(* CoDeSys 2.3.9.62 project: Ascensor_con_memoria_puerta_emergencia.pro *)
(* Libraries: Standard.lib 2.6.14 10:37:46, IecSfc.lib 2.6.14 11:37:46 *)

(* Global variable list: Global_Variables *)
VAR_GLOBAL
   (*Entradas *)

      (* Sensores de posición en plantas *)
      S0_1: BOOL;
      S1_1: BOOL;
      S2_1: BOOL;
      S3_1: BOOL;
      S0_2: BOOL;
      S1_2: BOOL;
      S2_2: BOOL;
      S3_2: BOOL;
      (* Pulsadores de llamadas en planta *)
      P0: BOOL;
      P1: BOOL;
      P2: BOOL;
      P3: BOOL;
    (* Pulsadores en cabina  *)
      C0_1: BOOL;
      C1_1: BOOL;
      C2_1: BOOL;
      C3_1: BOOL;
      C0_2: BOOL;
      C1_2: BOOL;
      C2_2: BOOL;
      C3_2: BOOL;
   (*Salidas *)
      Motor_arriba_1 : BOOL;
      Motor_Abajo_1 : BOOL;
     Motor_arriba_2 : BOOL;
      Motor_Abajo_2 : BOOL;
   (* luces asociadas a los pulsadores. Se usarán
        si se quiere implementar memoria de llamada *)
     LuzP0:BOOL;
     LuzP1:BOOL;
     LuzP2:BOOL;
     LuzP3:BOOL;
     LuzC0_1:BOOL;
     LuzC1_1:BOOL;
     LuzC2_1:BOOL;
     LuzC3_1:BOOL;
     LuzC0_2:BOOL;
     LuzC1_2:BOOL;
     LuzC2_2:BOOL;
     LuzC3_2:BOOL;
(* otras variables*)
	Emergencia: BOOL;
	EmerBTN:BOOL;
	LuzEmer:BOOL;
	Rearme:BOOL;
	puerta:BOOL;
END_VAR

(* POU PLC_PRG, ST *)
PROGRAM PLC_PRG
VAR
END_VAR
Movimiento1;
Ascensor;
END_PROGRAM

(* POU Movimiento1, ST *)
PROGRAM Movimiento1
VAR
    pos1:INT:=0;
END_VAR
IF (Motor_arriba_1 AND pos1>=-240) THEN
   pos1:=pos1-2;
END_IF


IF (Motor_abajo_1 AND pos1<=-2) THEN
   pos1:=pos1+2;
END_IF

IF (pos1>=0 AND pos1<=2) THEN
  S0_1:=TRUE;
ELSE
  S0_1:=FALSE;
END_IF

IF (pos1>=-78 AND pos1<=-74) THEN
  S1_1:=TRUE;
ELSE
  S1_1:=FALSE;
END_IF

IF (pos1>=-156 AND pos1<=-152) THEN
  S2_1:=TRUE;
ELSE
  S2_1:=FALSE;
END_IF

IF (pos1>=-242 AND pos1<=-240) THEN
  S3_1:=TRUE;
ELSE
  S3_1:=FALSE;
END_IF
END_PROGRAM

(* POU Ascensor, SFC *)
PROGRAM Ascensor
VAR
	CicloInicial: BOOL := TRUE;
	luzInt: ARRAY [0..3]  OF BOOL;
	luzext: ARRAY [0..3]  OF BOOL;
	cola: ARRAY [0..4]  OF  BOOL; (* Si la posicion i está a true hay que ir a esa planta *)
	Sentido: BOOL:=TRUE;
	PlantaActual:INT:=0;
	encontrado:BOOL; (* Intero a bool*)
	PD:PlantaDec;
	i: INT; (*interno a seleccion*)
	FRear: F_TRIG;
	REmer: R_TRIG;
	PP: PulsaPlanta;
END_VAR
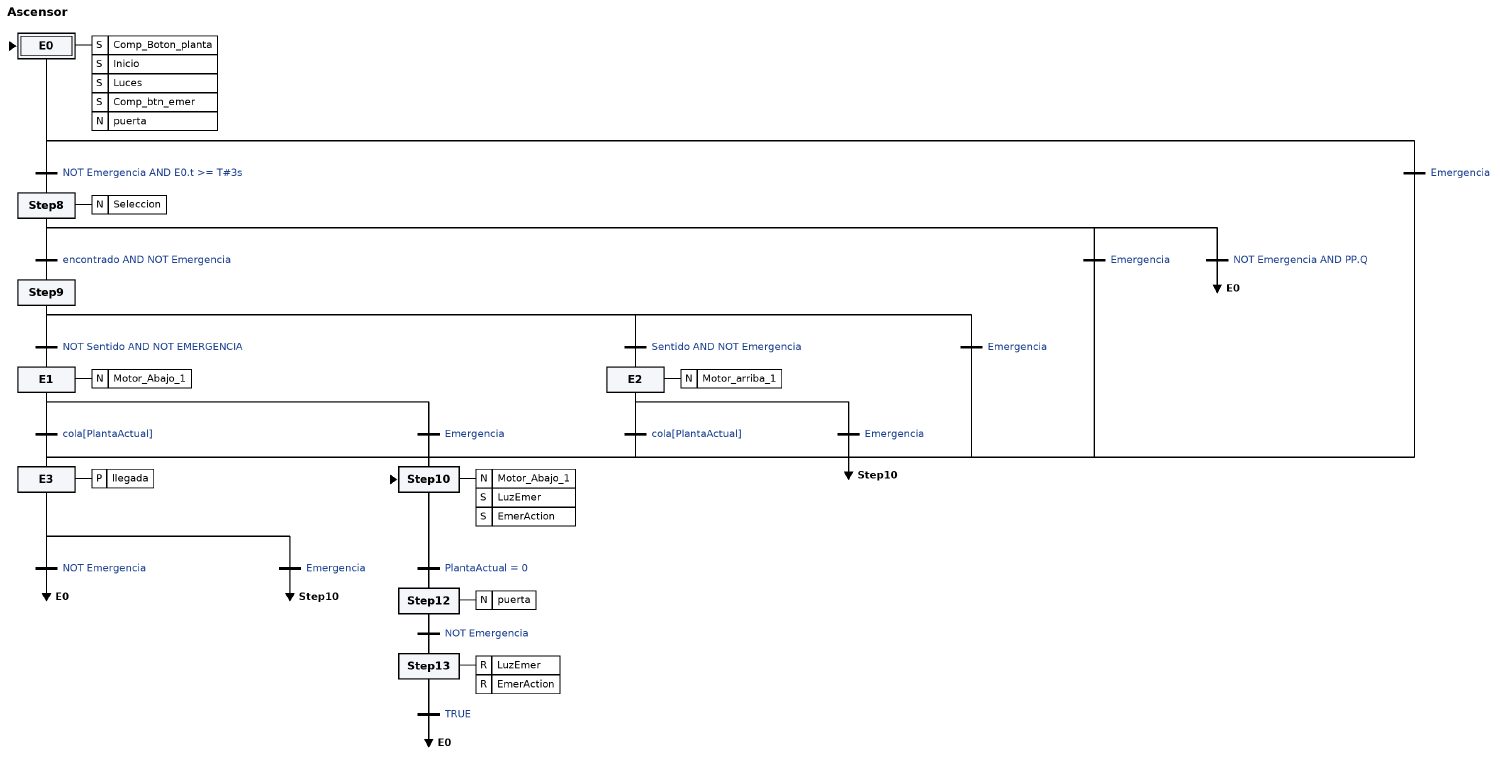
INITIAL_STEP E0:
	Comp_Boton_planta(S);
	Inicio(S);
	Luces(S);
	Comp_btn_emer(S);
	puerta(N);
END_STEP
TRANSITION FROM E0 TO Step8 := NOT Emergencia AND E0.t >= T#3s;
END_TRANSITION
TRANSITION FROM E0 TO Step10 := Emergencia;
END_TRANSITION
STEP Step8:
	Seleccion(N);
END_STEP
TRANSITION FROM Step8 TO Step9 := encontrado AND NOT Emergencia;
END_TRANSITION
TRANSITION FROM Step8 TO Step10 := Emergencia;
END_TRANSITION
TRANSITION FROM Step8 TO E0 := NOT Emergencia AND PP.Q;
END_TRANSITION
STEP Step9:
END_STEP
TRANSITION FROM Step9 TO E1 := NOT Sentido AND NOT EMERGENCIA;
END_TRANSITION
TRANSITION FROM Step9 TO E2 := Sentido AND NOT Emergencia;
END_TRANSITION
TRANSITION FROM Step9 TO Step10 := Emergencia;
END_TRANSITION
STEP E1:
	Motor_Abajo_1(N);
END_STEP
TRANSITION FROM E1 TO E3 := cola[PlantaActual];
END_TRANSITION
TRANSITION FROM E1 TO Step10 := Emergencia;
END_TRANSITION
STEP Step10:
	Motor_Abajo_1(N);
	LuzEmer(S);
	EmerAction(S);
END_STEP
TRANSITION FROM Step10 TO Step12 := PlantaActual = 0;
END_TRANSITION
STEP Step12:
	puerta(N);
END_STEP
TRANSITION FROM Step12 TO Step13 := NOT Emergencia;
END_TRANSITION
STEP Step13:
	LuzEmer(R);
	EmerAction(R);
END_STEP
TRANSITION FROM Step13 TO E0 := TRUE;
END_TRANSITION
STEP E2:
	Motor_arriba_1(N);
END_STEP
TRANSITION FROM E2 TO E3 := cola[PlantaActual];
END_TRANSITION
TRANSITION FROM E2 TO Step10 := Emergencia;
END_TRANSITION
STEP E3:
	llegada(P);
END_STEP
TRANSITION FROM E3 TO E0 := NOT Emergencia;
END_TRANSITION
TRANSITION FROM E3 TO Step10 := Emergencia;
END_TRANSITION
END_PROGRAM
ACTION Comp_Boton_planta:
(* Se encarga de  la  pulsacion de los botones  *)
(* no se puede añadir una planta a la memoria si ya estoy parado  en ella o hay una emergencia *)
IF NOT ( Emergencia OR (S0_1 AND NOT Motor_Abajo_1 AND NOT Motor_arriba_1) )AND (C0_1 OR  P0) THEN
cola[0]:= TRUE;
luzint[0]:= C0_1 OR luzInt[0];
luzext[0]:= P0 OR luzext[0];
ELSIF NOT( Emergencia OR (S1_1 AND NOT Motor_Abajo_1 AND NOT Motor_arriba_1)) AND (C1_1 OR  P1) THEN
cola[1]:= TRUE;
luzint[1]:= C1_1 OR luzInt[1];
luzext[1]:= P1 OR luzext[1];
ELSIF NOT( Emergencia OR (S2_1 AND NOT Motor_Abajo_1 AND NOT Motor_arriba_1) ) AND (C2_1 OR  P2) THEN
cola[2]:= TRUE;
luzint[2]:= C2_1 OR luzInt[2];
luzext[2]:= P2 OR luzext[2];
ELSIF NOT (Emergencia OR (S3_1 AND NOT Motor_Abajo_1 AND NOT Motor_arriba_1)) AND (C3_1 OR  P3) THEN
cola[3]:= TRUE;
luzint[3]:= C3_1 OR luzInt[3];
luzext[3]:= P3 OR luzext[3];
END_IF
END_ACTION
ACTION Comp_btn_emer:
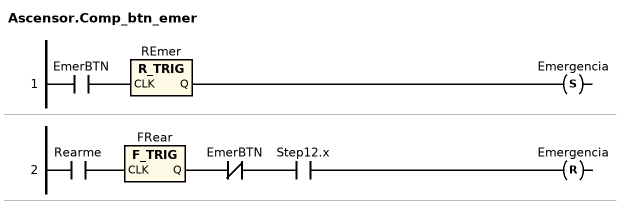
_LD_ (* Ladder Diagram *)
NETWORK 1
	[EmerBTN] - REmer:R_TRIG(CLK: *) --- (S Emergencia)
NETWORK 2
	[Rearme] - FRear:F_TRIG(CLK: *) - [/EmerBTN] - [Step12.x] --- (R Emergencia)
_END_LD_
(* the same logic as Structured Text *)
(* Network 1 *)
REmer(CLK := EmerBTN);
IF REmer.Q THEN Emergencia := TRUE; END_IF;
(* Network 2 *)
FRear(CLK := Rearme);
IF FRear.Q AND NOT EmerBTN AND Step12.x THEN Emergencia := FALSE; END_IF;
END_ACTION
ACTION EmerAction:
(* apagamos las luces de los pulsadores, vaciamos la cola y la planta destino*)
luzInt[0] := FALSE;

luzInt[1] := FALSE;

luzInt[2] := FALSE;

luzInt[3] := FALSE;


luzext[0] := FALSE;

luzext[1] := FALSE;

luzext[2] := FALSE;

luzext[3] := FALSE;


cola[0] := FALSE;

cola[1] := FALSE;

cola[2] := FALSE;

cola[3] := FALSE;

cola[4] := FALSE;

Sentido:=FALSE;
encontrado:=FALSE;
END_ACTION
ACTION inicio:
PD(SP0:=S0_1,SP1:=S1_1,SP2:=S2_1,SP3:=S3_1,PAct=>PlantaActual);
PP(SP0:=S0_1,SP1:=S1_1,SP2:=S2_1,SP3:=S3_1, PC0:=C0_1,PC2:=C2_1,PC3:=C3_1,PC1:=C1_1,PE0:=P0,PE1:=P1, PE2:=P2, PE3:=P3);
END_ACTION
ACTION llegada:
(* quitamos la planta cacutal de la cola*)
IF NOT (PlantaActual = 4) THEN
cola[PlantaActual]:= FALSE;
luzext[PlantaActual]:=FALSE;
luzint[PlantaActual]:=FALSE;
encontrado:= FALSE;
END_IF
END_ACTION
ACTION Luces:
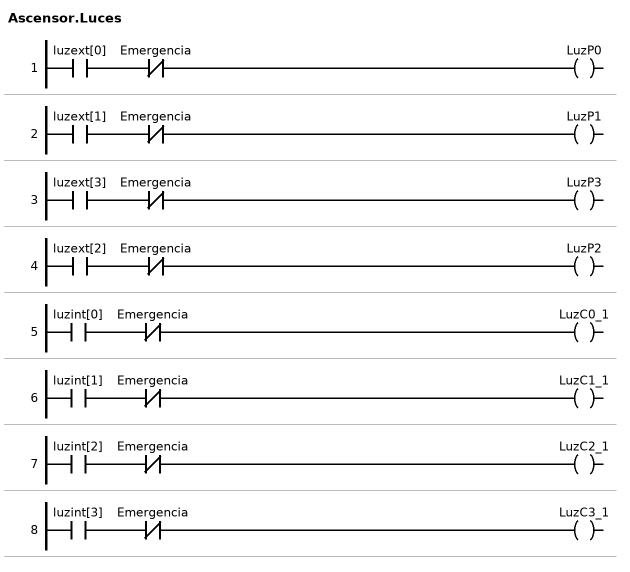
_LD_ (* Ladder Diagram *)
NETWORK 1
	[luzext[0]] - [/Emergencia] --- (LuzP0)
NETWORK 2
	[luzext[1]] - [/Emergencia] --- (LuzP1)
NETWORK 3
	[luzext[3]] - [/Emergencia] --- (LuzP3)
NETWORK 4
	[luzext[2]] - [/Emergencia] --- (LuzP2)
NETWORK 5
	[luzint[0]] - [/Emergencia] --- (LuzC0_1)
NETWORK 6
	[luzint[1]] - [/Emergencia] --- (LuzC1_1)
NETWORK 7
	[luzint[2]] - [/Emergencia] --- (LuzC2_1)
NETWORK 8
	[luzint[3]] - [/Emergencia] --- (LuzC3_1)
_END_LD_
(* the same logic as Structured Text *)
(* Network 1 *)
LuzP0 := luzext[0] AND NOT Emergencia;
(* Network 2 *)
LuzP1 := luzext[1] AND NOT Emergencia;
(* Network 3 *)
LuzP3 := luzext[3] AND NOT Emergencia;
(* Network 4 *)
LuzP2 := luzext[2] AND NOT Emergencia;
(* Network 5 *)
LuzC0_1 := luzint[0] AND NOT Emergencia;
(* Network 6 *)
LuzC1_1 := luzint[1] AND NOT Emergencia;
(* Network 7 *)
LuzC2_1 := luzint[2] AND NOT Emergencia;
(* Network 8 *)
LuzC3_1 := luzint[3] AND NOT Emergencia;
END_ACTION
ACTION Seleccion:
(* Selecciona la planta segun la planta actual *)
    IF sentido AND NOT (PlantaActual=3) THEN (* Subida *)
        FOR i := PlantaActual + 1 TO 3 DO
            IF cola[i] THEN
                 encontrado:=TRUE;

                EXIT;
            END_IF;
        END_FOR;
    ELSIF NOT (PlantaActual=0) AND NOT Sentido THEN
        FOR i := PlantaActual - 1 TO 0 BY -1 DO
            IF cola[i] THEN
                encontrado:=TRUE;

                EXIT;
            END_IF;
        END_FOR;
    END_IF;

    (* Si no encontró, cambiar el sentido y repetir la búsqueda *)
    IF  NOT  encontrado THEN
        sentido := NOT sentido;

        IF sentido AND NOT (PlantaActual=3)  THEN (* Subida *)
            FOR i := PlantaActual + 1 TO 3 DO
                IF cola[i] THEN
                     encontrado:=TRUE;
                    EXIT;
                END_IF;
            END_FOR;
        ELSIF NOT (PlantaActual=0) AND NOT Sentido THEN
            FOR i := PlantaActual - 1 TO 0 BY -1 DO
                IF cola[i] THEN
                     encontrado:=TRUE;
                    EXIT;
                END_IF;
            END_FOR;
        END_IF;
    END_IF;
END_ACTION

(* POU PlantaDec, ST *)
FUNCTION_BLOCK PlantaDec
VAR_INPUT
	SP0:BOOL;
	SP1:BOOL;
	SP2:BOOL;
	SP3:BOOL;
END_VAR
VAR_OUTPUT
	PAct:INT;
END_VAR
VAR

END_VAR
(*Decodificador de planta*)
IF SP0 THEN
PAct :=0;
ELSIF SP1 THEN
PAct:=1;
ELSIF Sp2 THEN
Pact:=2;
ELSIF SP3 THEN
Pact:=3;
ELSE PACT:= 4 ;
END_IF
END_FUNCTION_BLOCK

(* POU PulsaPlanta, LD *)
FUNCTION_BLOCK PulsaPlanta
VAR_INPUT
	SP0,Sp1,sp2,sp3: BOOL; (*sensores de planta*)
	PC0,PC1,PC2,PC3: BOOL;(*pulsadores de cabina*)
	PE0,PE1,PE2,pE3:BOOL; (* pulsadores  externos*)
END_VAR
VAR_OUTPUT
	Q:BOOL:=FALSE;
END_VAR
VAR
END_VAR
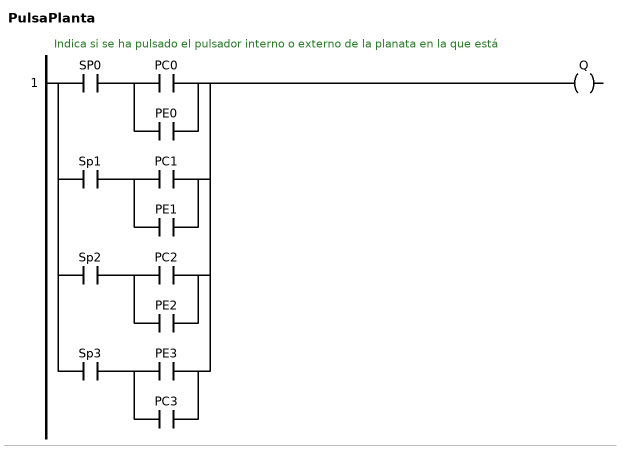
_LD_ (* Ladder Diagram *)
NETWORK 1 (* Indica si se ha pulsado el pulsador interno o externo de la planata en la que está *)
	{ [SP0] - { [PC0] | [PE0] } | [Sp1] - { [PC1] | [PE1] } | [Sp2] - { [PC2] | [PE2] } | [Sp3] - { [PE3] | [PC3] } } --- (Q)
_END_LD_
(* the same logic as Structured Text *)
(* Network 1: Indica si se ha pulsado el pulsador interno o externo de la planata en la que está *)
Q := SP0 AND (PC0 OR PE0) OR Sp1 AND (PC1 OR PE1) OR Sp2 AND (PC2 OR PE2) OR Sp3 AND (PE3 OR PC3);
END_FUNCTION_BLOCK

(* Visualisation Ascensor
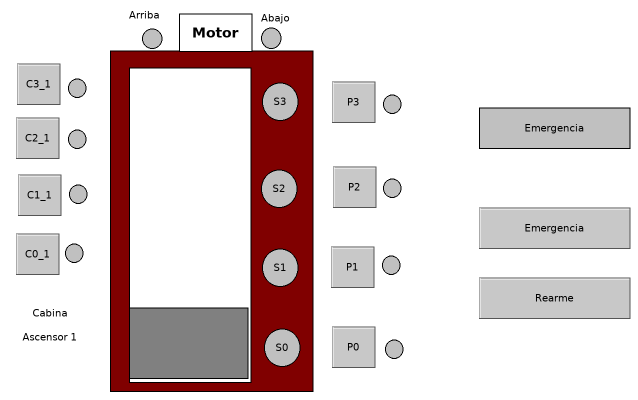
ellipse at (285,341)-(321,379): text "S0"; alarm colour if S0_1
ellipse at (283,261)-(319,299): text "S1"; alarm colour if S1_1
ellipse at (282,182)-(318,220): text "S2"; alarm colour if S2_1
ellipse at (283,95)-(319,133): text "S3"; alarm colour if S3_1
rounded rectangle at (150,320)-(269,391): alarm colour if puerta; y offset Movimiento1.pos1
button at (353,339)-(396,380): text "P0"; taps P0
button at (352,259)-(395,300): text "P1"; taps P1
button at (354,179)-(397,220): text "P2"; taps P2
button at (353,94)-(396,135): text "P3"; taps P3
rectangle at (200,26)-(273,64): text "Motor"
ellipse at (163,41)-(183,61): alarm colour if Motor_arriba_1
ellipse at (282,40)-(302,61): alarm colour if Motor_abajo_1
rectangle at (138,18)-(193,37): text "Arriba"
rectangle at (269,21)-(324,40): text "Abajo"
button at (37,246)-(80,287): text "C0_1"; taps C0_1
button at (39,187)-(82,228): text "C1_1"; taps C1_1
button at (37,130)-(80,171): text "C2_1"; taps C2_1
button at (38,76)-(81,117): text "C3_1"; taps C3_1
rectangle at (28,305)-(114,346): text "Cabina"
rectangle at (28,329)-(114,370): text "Ascensor 1"
ellipse at (89,91)-(107,110): alarm colour if LuzC3_1
ellipse at (89,142)-(107,161): alarm colour if LuzC2_1
ellipse at (90,197)-(108,216): alarm colour if LuzC1_1
ellipse at (86,256)-(104,275): alarm colour if LuzC0_1
ellipse at (404,107)-(422,126): alarm colour if LuzP3
ellipse at (404,191)-(422,210): alarm colour if LuzP2
ellipse at (403,268)-(421,287): alarm colour if LuzP1
ellipse at (406,352)-(424,371): alarm colour if LuzP0
rectangle at (500,120)-(651,161): text "Emergencia"; alarm colour if LuzEmer
button at (500,220)-(651,261): text "Emergencia"; taps EmerBTN
button at (500,290)-(651,331): text "Rearme"; taps Rearme
3 more shapes without text or variables
*)
